Staubli VAL3: DismountGripper.pgx

program DismountGripper()
begin
  sInfo="Parking gripper..."
        movej(jChange,tChanger,mNomSpeed)

        bOk=watch(bTUnlocked==false and bTLocked==true,5)

        if bOk==true
          movej(appro(pTool1,{0,0,-200,0,0,0}),tChanger,mChange)
          waitEndMove()
          movel(pTool1,tChanger,mAppro)

          bOk=watch(bEstPinza==true,20)
          if bOk==true
            dChangerValve=true
            delay(0.1)
            bOk=watch(bTUnlocked==true and bTLocked==false,30)
            //5
            if bOk==true
              movel(appro(pTool1,{0,0,-100,0,0,0}),tChanger,mChange)
              bOk=watch(bHerramientaRobot==false,5)
              if bOk==true
                movej(jChange,tChanger,mNomSpeed)
                waitEndMove()

              else
                disablePower()
                userPageAlert("Error. Check parking station.")
                bError=true

              endIf

            else
              disablePower()
              userPageAlert("Error. Tool can not be unlocked, check neumatic circuit.")
              bError=true

            endIf

          else
            disablePower()
            userPageAlert("Error. Tool not detected at parking station")
            bError=true

          endIf

        else
          disablePower()
          userPageAlert("Error. Tool can not be unlocked, check neumatic circuit")
          bError=true

        endIf
end
